// TIA Portal V18 export
TYPE "ProcessCheck_ShW"
// stored: IsFailsafeCompliant false
   STRUCT
      Trigger : Bool;
      Mode : String[48];
      Result : Int;
      Completed : Bool;
   END_STRUCT;
END_TYPE
